(*
Nazwa:			FB_RollerScrewer
Opis:			Zakręcarka rolkowa
Wersja:			v0.5
Data:			2020-03-16
Autor:			DP
Urzadzenia:		Serwo zakręcania, podnosnik JIESANG, rolki, docisk z góry
Konfiguracja:	
Info:  
- ZMIANA ESTOP - blad w trybie manualnym po ESTOPIE
- Dddano kasowanie ruchów w górę po błędzie
- Dodano opisy błędów serwa
- Dodano błędy od nastaw powyżej max i min (error 7 i 8)
- Zmiana Homingów według CatchStation
- zmiana momentu zacisniecia rolek
*)

FUNCTION_BLOCK FB_RollerScrewer
VAR_INPUT
	bEnable:BOOL;						//Zezowlenie na pracę zakręcarki rolkowej
	bEStop:BOOL;						//Stop awaryjny nieaktywny
	bRun:BOOL;							//Rozkaz zakręcania 
	bHoming:BOOL;						//Zezwolenie na wykonanie bazowania i pozycjonowania zakręcarki rolkowej
	bHeightSet:BOOL;					//Ustaw wysokość
	bIgnoreError:BOOL;					//Ignorowania błędów cyklu pracy
	bReset:BOOL;						//Reset błędu, jeśli w stanie "eError"
	nPositionHeightSV:LREAL;			//Wysokość zadana na której ma znajdować się zakręcarka rolkowa
	lrMaxHeight:LREAL;					//Maksymalna wysokość zakręcarki rolkowej
	lrMinHeight:LREAL;					//Minimalna wysokość zakręcarki rolkowej
	iScrewerSetTorque:INT;				//Zadany moment dokręcania [%]
	iScrewTightTime:INT;				//Czas przytrzymania po uzyskaniu momentu [ms] 
	lrScrewerAcceleration:LREAL;			//Przyspieszenie zakręcarki rolkowej
	lrScrewerDeceleration:LREAL;			//Opóźnienie zakręcarki rolkowej
	lrScrewerSpeed:LREAL;				//Prędkość zakręcarki rolkowej
	lrFindigScrewDegree:LREAL;			//Kąt wycofania zakręcarki rolkowej przy szukaniu gwintu
	lrScrewerFrontActualTorque:LREAL;			//Aktualny moment [%]
	lrScrewerRearActualTorque:LREAL;			//Aktualny moment [%]
	rRearActualMotorTemperature :REAL;	// Aktualna temperatura silnika tylniego
	rFrontActualMotorTemperature :REAL;	// Aktualna temperatura silnika tylniego
	bRollsPressedSensor: BOOL; 			// Wejście czujnika zaciśnięcie rolek zakręcarki
	bRollsUnPressedSensor: BOOL; 		// Wejście czujnika odpuszczenia rolek zakręcarki
	bUnPressedTopSensor: BOOL;			// Wejscie czujnika wycofania docisku górnego zakręcarki rolkowej
	lrManualOverride:LREAL;				// Procentowa redukcja prędkości wszystkich serw (Tylko w trybie manualnym)
	bManualMovement:BOOL; 			// Uruchomienie trybu ruchów ręcznych
	bFindingScrewBeginingOption:BOOL; 	//OPCJA. Szukaj początku gwintu nakrętki i opakowania. Zakręcarka napjpierw obraca się w lewo, a po znalezienu gwintu przystepuje do zakręcania;
	nTopActuatorTimeDelayOff:UINT;  	//czas po którym odpusczany jest docisk górny
	bUnlockColision:BOOL:=FALSE;		//Odblokowywanie możliwośći kolizji

	_HEIGHTMOTOR_ :BOOL;	
	bHeightMotorEncoderPulse :BOOL;			//Sygnał impulsów enkodera siłownika
	rHeightMotorPositionOffset :REAL;		//Wysokość bazowani podnośnika
	
	_ALARMINFO_ :BOOL;
	iStationIndex:UDINT;				//Numer stacji 
	sStationName:STRING;				//Nazwa stacji	
	
END_VAR
VAR_OUTPUT
	eState: E_Station;				// Stan zakręcarki rolkowej
	eRunningState:E_RollerScrewer;	// Stan zakręcarki	
	bError: BOOL;					// Błąd stacji
	udiErrorID: UDINT;				// Nr błędu zakręcarki rolkowej
	sErrorDescription:STRING(200);	// Opis błędu
	sErrorDescription2: STRING(200);// Opis błędu
	sErrorStationName: STRING;		// Nazwa stacj
	nScrewingServoErrorNr: UDINT;	// Nr błędu serwo zakręcarki
	bPressingTopActuator: BOOL; 	// Sterowanie zaworem dociskania nakrętki zaciskarki rolkowej od góry
	bPressingRollsActuator: BOOL; 	// Sterowanie zaworem dociskania rolek od boku
	bHeightMotorUp:BOOL;			// Sterowanie silnikiem podnośnika  - RUCH W GÓRĘ
	bHeightMotorDown:BOOL;			// Sterowanie silnikiem podnośnika  - RUCH W DÓŁ
	lrHeightMotorCV:LREAL;			// Aktualna pozycja podnośnika
	uiScrewingFrontTorqueControl:UINT;	// Kontola momentu zakręcania	
	uiScrewingRearTorqueControl:UINT;	// Kontola momentu zakręcania	

	bWarning: BOOL;
	udiWarningID: UDINT;
	tCycleTime:TIME;		
	bHomingDone:BOOL;				// Wymagane ponowne bazowanie (blad podczas bazowania lub stop awaryjny)
	bCycleDone:BOOL;
	bCycleNotDone:BOOL;		
	bAdjustingTorqueDone:BOOL;
	iAdjustingTorque:INT;
	lrAdjustingMaxTorque: LREAL;
END_VAR

VAR
	tonHeightNoChange: TON; // Timer wykrycia braku ruchu siłownika zmiany wysokości stacji
	nLastPositionHeightCV: LREAL;// Pozycja podnośnika w poprzednim cyklu programu
	tonErrorHeightChange: TON; // Timer błędu podnośnika
	rtEncoderHomed:R_TRIG;
	tonCycleTimer:TON;
	rtrigCycleTimerRead:R_TRIG;
	
	mcScrewerFrontMoveVelocity		:MC_MoveVelocity; 	// Ruch prędkościowy
	mcScrewerFrontHalt				:MC_HALT; 			// Zatrzymanie zakręcania
	mcScrewerFrontManualMove		:MC_JOG; 			// Blok obrotu ręcznego zakręcarką
	mcScrewerFrontStop				:MC_Stop; 			// Trwałe zatrzymywanie Serwo
	mcScrewerFrontPower				:MC_POWER; 			// Zasilanie napędu zakręcarki
	fbScrewerFrontHardReset			:FB_SoEReset;
	mcScrewerFrontSoftReset			:MC_Reset;
	mcScrewerFrontSetPosition		:MC_SetPosition;
	mcScrewerFrontMoveRelative		:MC_MoveRelative;

	mcScrewerRearMoveVelocity		:MC_MoveVelocity; 	// Ruch prędkościowy
	mcScrewerRearHalt				:MC_HALT; 			// Zatrzymanie zakręcania
	mcScrewerRearManualMove			:MC_JOG; 			// Blok obrotu ręcznego zakręcarką
	mcScrewerRearStop				:MC_Stop; 			// Trwałe zatrzymywanie Serwo
	mcScrewerRearPower				:MC_POWER; 			// Zasilanie napędu zakręcarki
	fbScrewerRearHardReset			:FB_SoEReset;
	mcScrewerRearSoftReset			:MC_Reset;
	mcScrewerRearSetPosition		:MC_SetPosition;
	mcScrewerRearMoveRelative		:MC_MoveRelative;
	
	bScrewFound: BOOL; //Zakręcarka znalazła początek gwintu
	nMaxTorque: LREAL; //Maksymalny moment podczas szukania poczatku gwintu
	nMinTorque: LREAL; // Najmniejszy moment podczas szukania poczatku gwintu

	tonTightScrewingTimer: TON; // Timer potwierdzenia dokręcenia nakrętki
	bScrewed: BOOL; // Nakrętka zakręcona

	tonTooLongScrewing: TON; // Błąd zbyt długiego zakręcania

	bScrewerFrontServoPower: BOOL; // Zmienna sterujaca zasilaniem serwo Zakręcark
	bScrewerRearServoPower: BOOL; // Zmienna sterujaca zasilaniem serwo Zakręcark

	// Za długie szukanie gwintu
	tonTooLongFinding: TON;
	tonPosDiffError	:TON;
	bStopped: BOOL;
	// Ustawianie pozycji napedu zakrecającego po zakręceniu nakrętki


	// Pozycja rozpoczęcia zakrecania
	lrStartScrewingPos: LREAL;
	
	// Ruch relatywny zakręcarki

	lrStartPositionScrewerFront: LREAL;
	lrStartPositionScrewerRear: LREAL;	
	tonPressingTopDelay: TON;
	tonPressingRollsDelay: TON;
	tonUpPressRollsDelay: TON;
	tonPressingRollsReliseDelay: TON;
	tonTopActuatorDelayOff: TON;
	tonPushingCapDelay: TON;
	tonRollsPressedDelay: TON;
	tofMotorUpPermition: TOF;
	tofMotorDownPermition: TOF;
	tonLimitPosMinReachedDelay: TON;
	tonLimitPosMaxReachedDelay: TON;
	tonMaxHeight: TON;

	bStateError: BOOL;

	//Podnośnik Jiesang	
	fbHeightMotorEncoder			:FB_JiesangActuatorEncoder;	// Blok enkodera podnośnika chwytaka stabilizującego pod zakręcarką	
	bHeightMotorEncoderCounterReset	:BOOL; 						// Sygnał resetu enkodera
	bHeightMotorEncoderHomed		:BOOL;						// Informacja od enkodera że jest zbazowany

	eLastState						:E_Station;			// Stan ogólny bloku
	eLastRunningState				:E_RollerScrewer;	// Stan podbloku
	eLastStateTemp					:E_Station;			// Stan ogólny bloku
	eLastRunningStateTemp			:E_RollerScrewer;	// Stan podbloku	
	sWarningDescription				:STRING;
	
	nCaseAdjustingTorque: INT;
	tonAdjustingTightScrewingTimer: TON;
	tonAdjustingGripperClose: TON;
	uiAdjustingScrewerTorqueControl: UINT;
	bAdjustingScrewed: BOOL;
	tonAdjustingCase40: TON;
	bAdjustingSetTorqueAchieved: BOOL;
	bAdjustingTorqueTooHigh: BOOL;
	bAdjustingTorqueTooLow: BOOL;
	lrMotorNominalTorque: LREAL;
	lrScrewerActualTorqueNm: LREAL;
	
	tonDelayServoOn			: TON;

	tonRearActualMotorTemperatureTooHigh: TON;
	tonFrontActualMotorTemperatureTooHigh: TON;
END_VAR

VAR_IN_OUT
	bManualPressingTopActuator		:BOOL;		// Sterowanie w trybie serwisowym zaworem dociskania nakrętki zaciskarki rolkowej od góry
	bManualPressingRollsActuator	:BOOL;		// Sterowanie w trybie serwisowym zaworem dociskania rolek od boku
	bManualHeightMotorUp			:BOOL;		// Ruch ręczny podnośnika stacji w górę
	bManualHeightMotorDown			:BOOL;		// Ruch ręczny podnośnika stacji w dół
	bManualScrewClockwise			:BOOL;		// Ruch ręczny zakręcarką w kierunku wskazówek zegara;
	bManualScrewCClockwise			:BOOL;		// Ruch ręczny zakręcarką w kierunku przeciwnym do wskazówek zegara;
	RollerScrewerFrontAxisRef		:AXIS_REF;	// Struktura sterowania NC dla serwa zakręcania
	RollerScrewerRearAxisRef		:AXIS_REF;	// Struktura sterowania NC dla serwa zakręcania	

END_VAR

(*Przepisywanie Homingu , rozdzielenie wyjść*)

HeightMotor();
ErrorHandling();
Control();
ServoFrontControlBlocks();
ServoRearControlBlocks();
Statistics();

(*Zapisywanie ostatniego stanu*)
IF eLastStateTemp<>eState THEN
	eLastState := eLastStateTemp;
END_IF
eLastStateTemp := eState;
IF eLastRunningStateTemp<>eRunningState THEN
	eLastRunningState := eLastRunningStateTemp;
END_IF
eLastRunningStateTemp := eRunningState;
(*Koniec Zapisywanie ostatniego stanu*)


nLastPositionHeightCV:=lrHeightMotorCV;

ACTION Control:
	(** TIMERY**)
	rtEncoderHomed				(CLK:= bHeightMotorEncoderHomed,Q=>);
	tonHeightNoChange			(IN:= ((bHeightMotorUp OR bHeightMotorDown) AND (nLastPositionHeightCV=lrHeightMotorCV)), PT:= T#1S); 
	tonLimitPosMinReachedDelay	(IN:= (lrHeightMotorCV<=lrMinHeight) AND eState=E_Station.eHoming,PT:= T#2S);
	tonLimitPosMaxReachedDelay	(IN:= (lrHeightMotorCV>=lrMaxHeight) AND eState=E_Station.eHoming,PT:= T#2S);

	tonPressingRollsReliseDelay(IN:= NOT bPressingRollsActuator AND NOT bPressingTopActuator, PT:= T#40MS);	
	tonTightScrewingTimer		(IN:= (eRunningState=E_RollerScrewer.eScrewing) AND 
								NOT tonTightScrewingTimer.Q AND mcScrewerFrontMoveVelocity.Execute AND mcScrewerRearMoveVelocity.Execute AND 
								((lrScrewerFrontActualTorque>=iScrewerSetTorque) OR (lrScrewerRearActualTorque>=iScrewerSetTorque)) AND 
								ABS(RollerScrewerFrontAxisRef.NcToPlc.PosDiff)>360 AND ABS(RollerScrewerRearAxisRef.NcToPlc.PosDiff)>360 
								AND NOT bScrewed ,PT:= INT_TO_TIME(iScrewTightTime));
	tonTopActuatorDelayOff		(IN:= bPressingTopActuator AND eRunningState=E_RollerScrewer.eScrewing, PT:= UINT_TO_TIME(nTopActuatorTimeDelayOff));	
	tonPushingCapDelay			(IN:= (eRunningState=E_RollerScrewer.ePushingCap) AND (NOT bUnPressedTopSensor OR  nTopActuatorTimeDelayOff=0), PT:= T#100MS);
	tonRollsPressedDelay		(IN:= (eRunningState=E_RollerScrewer.ePushingCap) AND NOT bRollsUnpressedSensor, PT:= T#0MS); //bylo 200

	tonDelayServoOn				(IN:=(eState = E_Station.ePreparingToReady), PT:=T#2S);
	
	(*****Wyłączenie enable*****)
	IF NOT bEnable THEN
		IF eState <> E_Station.eDisabled AND eState <> E_Station.ePreparingToDisable THEN
				eState 								:= E_Station.ePreparingToDisable; 
		END_IF	
	END_IF

	(*****Estop*****)
	IF NOT bEstop  THEN	
		IF eState <> E_Station.eAborted AND eState <> E_Station.eAborting AND eState <> E_Station.eDisabled THEN
				eState 								:= E_Station.eAborting; 
		END_IF
	END_IF

	
	CASE eState OF
	/////////////////////////////	
		E_Station.eDisabled: 						// Stan nieaktywnosci (Stacja wyłączona) 
		
			IF bEnable THEN
				eState 								:= E_Station.ePreparingToReady; 
			END_IF 
			
    /////////////////////////////	    
		E_Station.eAborted: 						// Stan bezpiecznego zatrzymania (po Abortingu) 

			IF bEStop THEN
				eState 								:= E_Station.ePreparingToReady;
			END_IF
			
	/////////////////////////////	
		E_Station.eAborting:                 		// Stan bezpiecznego zatrzymywania (po EStopie)
		
			bHeightMotorDown		:=	FALSE;
			bHeightMotorUp			:=	FALSE;	
		
			bPressingTopActuator					:= FALSE;
			bPressingRollsActuator					:= FALSE;

			mcScrewerFrontPower.Override			:= 100;
			mcScrewerFrontStop.Execute				:= NOT bStopped;
			mcScrewerFrontMoveVelocity.Execute		:= FALSE;
			mcScrewerFrontManualMove.JogBackwards	:= FALSE;
			mcScrewerFrontManualMove.JogForward		:= FALSE;
			
			mcScrewerRearPower.Override				:= 100;
			mcScrewerRearStop.Execute				:= NOT bStopped;
			mcScrewerRearMoveVelocity.Execute		:= FALSE;
			mcScrewerRearManualMove.JogBackwards	:= FALSE;
			mcScrewerRearManualMove.JogForward		:= FALSE;
			
			IF ((mcScrewerFrontStop.Done OR NOT bScrewerFrontServoPower) AND (mcScrewerRearStop.Done OR NOT bScrewerRearServoPower)) OR bStopped THEN
				bStopped							:= FALSE;
				bScrewerFrontServoPower				:= FALSE;
				mcScrewerFrontStop.Execute			:= FALSE;
				bScrewerRearServoPower				:= FALSE;
				mcScrewerRearStop.Execute			:= FALSE;
				eState								:= E_Station.eAborted; 
				eRunningState						:= E_RollerScrewer.eReady;
			END_IF		
			
			
	/////////////////////////////			
		E_Station.eError:                 	 		// Stan błędu 	
				
			IF bReset THEN
				eState 								:= E_Station.eResetting;
			ELSE
				mcScrewerFrontSoftReset				(Execute:= FALSE,Axis:= RollerScrewerFrontAxisRef);	
				mcScrewerRearSoftReset				(Execute:= FALSE,Axis:= RollerScrewerRearAxisRef);	
			END_IF
			
	/////////////////////////////
		E_Station.eResetting:						// Stan resetowania bledu (po Errorze)
			
			//Procedura obsługi resetu w zależności od błędu
			CASE udiErrorID-iStationIndex OF
		
				//Error 1 - ZA DŁUGIE ZAKRĘCANIE	
				1:
					IF tonPressingRollsReliseDelay.Q AND RollerScrewerFrontAxisRef.Status.StandStill AND RollerScrewerRearAxisRef.Status.StandStill THEN
						;
						udiErrorID					:= 0;
						sErrorDescription			:= '';	
						bError 						:= FALSE;	
					END_IF
					
				//Error 2,4,5,6,7,8	
				2,4,5,6,7,8:   
					 bError 						:= FALSE;
					 udiErrorID						:= 0;
					 sErrorDescription				:= '';		
			
				//Error 3 - BŁĄD SERWA ZAKRĘCANIA
				3:	
					//fbScrewerHardReset			(Execute:= NOT mcHeightMoveAbsolute.Execute,Axis:= ScrewingAxisRef);
					mcScrewerFrontSoftReset			(Execute:= TRUE,Axis:= RollerScrewerFrontAxisRef);
					mcScrewerRearSoftReset			(Execute:= TRUE,Axis:= RollerScrewerRearAxisRef);
					IF NOT fbScrewerFrontHardReset.Busy AND NOT mcScrewerFrontSoftReset.Busy AND mcScrewerFrontPower.Status AND NOT RollerScrewerFrontAxisRef.Status.Error
					AND NOT fbScrewerRearHardReset.Busy AND NOT mcScrewerRearSoftReset.Busy AND mcScrewerRearPower.Status AND NOT RollerScrewerRearAxisRef.Status.Error  THEN
						fbScrewerFrontHardReset		(Execute:= FALSE,Axis:= RollerScrewerFrontAxisRef);
						fbScrewerRearHardReset		(Execute:= FALSE,Axis:= RollerScrewerRearAxisRef);
						mcScrewerFrontSoftReset		(Execute:= FALSE,Axis:= RollerScrewerFrontAxisRef);
						mcScrewerRearSoftReset		(Execute:= FALSE,Axis:= RollerScrewerRearAxisRef);
						bError 						:= FALSE;
						udiErrorID					:= 0;
						nScrewingServoErrorNr		:= 0;
						mcScrewerFrontPower.Override:= 100;
						mcScrewerRearPower.Override	:= 100;
						eState						:= E_Station.eReady;
						sErrorDescription			:= '';	
			
					ELSIF NOT fbScrewerFrontHardReset.Busy AND NOT mcScrewerFrontSoftReset.Busy AND NOT mcScrewerFrontPower.Status AND NOT bScrewerFrontServoPower AND NOT RollerScrewerFrontAxisRef.Status.Error
						AND NOT fbScrewerRearHardReset.Busy AND NOT mcScrewerRearSoftReset.Busy AND NOT mcScrewerRearPower.Status AND NOT bScrewerRearServoPower AND NOT RollerScrewerRearAxisRef.Status.Error THEN
						//fbScrewerHardReset(Execute:= FALSE,Axis:= ScrewingAxisRef);
						mcScrewerFrontSoftReset		(Execute:= FALSE,Axis:= RollerScrewerFrontAxisRef);
						mcScrewerRearSoftReset		(Execute:= FALSE,Axis:= RollerScrewerRearAxisRef);
						udiErrorID					:= 0;
						nScrewingServoErrorNr		:= 0;
						mcScrewerFrontPower.Override:= 100;
						mcScrewerRearPower.Override	:= 100;
						bError 						:= FALSE;
						sErrorDescription			:= '';
					END_IF		
					
			END_CASE	
			
			IF NOT bError THEN
				udiErrorID 							:= 	0;
   				sErrorDescription 					:= 	'';
	                                				
				eState 								:= 	E_Station.ePreparingToReady;
				mcScrewerFrontStop.Execute			:= FALSE;    
				mcScrewerRearStop.Execute			:= FALSE; 
			ELSE                    	
				eState 								:= 	E_Station.eError;
			END_IF
        
	/////////////////////////////
		E_Station.eManualMovement:     				// Stan ruchów manualnych  
       
			ManualMovements();
			//Wyjście z trybu serwisowego
			IF NOT bManualMovement THEN
				bManualPressingTopActuator			:= 	FALSE;
				bManualPressingRollsActuator		:= 	FALSE;
				bHeightMotorUp						:= 	FALSE;
				bHeightMotorDown					:= 	FALSE;
				mcScrewerFrontPower.Override			:= 	100;
				mcScrewerRearPower.Override			:= 	100;
				eState								:= 	E_Station.eReady;
			END_IF

	/////////////////////////////
		E_Station.eHoming:							// Stan bazowania 

			Homing();
			IF NOT bHoming AND NOT bHeightSet THEN
			   eState								:= 	E_Station.ePreparingToReady;
			   bHeightMotorUp						:= 	FALSE;
				bHeightMotorDown					:= 	FALSE;
			END_IF		
			
	/////////////////////////////
		E_Station.eHomingDone:                  	// Stan wykonania bazowania 

			bHeightMotorDown						:= 	FALSE;
			bHeightMotorUp							:= 	FALSE;
			bHeightMotorEncoderCounterReset			:= 	FALSE;
			bHomingDone								:= 	TRUE;
			IF NOT bHoming AND NOT bHeightSet THEN
			   	eState								:= 	E_Station.eReady;
			END_IF
			
	/////////////////////////////
		E_Station.ePreparingToReady:            	// Stan przygotowywania do gotowosci (zawsze przed Ready)  
	
			IF tonDelayServoOn.Q THEN
				bScrewerFrontServoPower				:= 	TRUE;
				bScrewerRearServoPower				:= 	TRUE;
			END_IF	

				
			bPressingTopActuator					:= 	FALSE;
			bPressingRollsActuator					:= 	FALSE;
			IF mcScrewerFrontPower.Status AND mcScrewerRearPower.Status THEN  	
				eState								:= 	E_Station.eReady;
				eRunningState						:= 	E_RollerScrewer.eReady;
			END_IF                              	
         	IF bIgnoreError THEN                	
				eState								:= 	E_Station.eReady;
				eRunningState						:= 	E_RollerScrewer.eReady;
			END_IF
	
	/////////////////////////////
		E_Station.ePreparingToDisable:         	 	// Stan przygotowywania do nieaktywnosci (po wyłączeniu Enable) 
  
			bScrewerFrontServoPower					:= 	TRUE;
			bScrewerRearServoPower					:= 	TRUE;

			
			bPressingTopActuator					:= 	FALSE;
			bPressingRollsActuator					:= 	FALSE;
			                        				
			bHeightMotorUp							:= 	TRUE;
			bHeightMotorDown						:= 	FALSE;
			IF tonHeightNoChange.Q THEN	
				bHeightMotorUp:= FALSE;
				IF  mcScrewerFrontPower.Status THEN
					bScrewerFrontServoPower			:= 	FALSE; //LU205
					bScrewerRearServoPower			:= 	FALSE;;//LU205
					eState							:= 	E_Station.eDisabled;
					eRunningState					:= 	E_RollerScrewer.eReady;
				END_IF
			END_IF				
         	IF bIgnoreError THEN
				bHeightMotorUp						:= 	FALSE;
				eState								:= 	E_Station.eDisabled;
				eRunningState						:= 	E_RollerScrewer.eReady;
			END_IF
			
	/////////////////////////////
		E_Station.eReady:							// Stan gotowosci 
		
			mcScrewerFrontStop.Execute:= FALSE;
		
			IF bRun AND NOT bCycleDone AND NOT bCycleNotDone THEN
				eState 								:= E_Station.eStarting; 
			END_IF
			IF bHoming OR bHeightSet THEN
				eState 								:= E_Station.eHoming; 
			END_IF
			IF bManualMovement THEN
				//Jeśli przejście w tryb ruchów manualnych przepisz wszystkie stany siłowników sterowanych przez moduł
				//aby zapobiec ewentualnym kolizjom po wejściu w tryb serwisowy
				bManualPressingTopActuator			:= 	bPressingTopActuator;
				bManualPressingRollsActuator		:= 	bPressingRollsActuator;
				bManualHeightMotorUp				:= 	bHeightMotorUp;
				bManualHeightMotorDown				:= 	bHeightMotorDown;
				mcScrewerFrontStop.Execute			:= 	FALSE;
				mcScrewerRearStop.Execute			:= 	FALSE;
				eState 								:= 	E_Station.eManualMovement; 
			END_IF
			IF NOT bRun THEN
				bCycleDone 							:= FALSE;
				bCycleNotDone 						:= FALSE;	
				bWarning							:= FALSE;	
			END_IF      

			bStopped								:= FALSE;
			mcScrewerFrontStop.Execute				:= FALSE;    
			mcScrewerRearStop.Execute				:= FALSE;                   			
			
	/////////////////////////////
		E_Station.eStopping:					// Stan zatrzymywania 
			
			Running();

			bPressingTopActuator					:= 	FALSE;
			bPressingRollsActuator					:= 	FALSE;
			
			mcScrewerFrontHalt.Execute				:= 	FALSE;			
			mcScrewerFrontStop.Execute				:= 	NOT bStopped;
			mcScrewerFrontMoveRelative.Execute		:= 	FALSE;
			mcScrewerFrontMoveVelocity.Execute		:= 	FALSE;
			uiScrewingFrontTorqueControl			:= 	0; // bylo 6000	
			mcScrewerFrontSoftReset					(Axis:= RollerScrewerFrontAxisRef, Execute:= TRUE);

			mcScrewerRearHalt.Execute				:= 	FALSE;			
			mcScrewerRearStop.Execute				:= 	NOT bStopped;
			mcScrewerRearMoveRelative.Execute		:= 	FALSE;
			mcScrewerRearMoveVelocity.Execute		:= 	FALSE;
			uiScrewingRearTorqueControl				:= 	0; // bylo 6000	
			mcScrewerRearSoftReset					(Axis:= RollerScrewerRearAxisRef, Execute:= TRUE);
			
			IF  (mcScrewerFrontStop.Done OR mcScrewerFrontStop.CommandAborted) AND 
				(mcScrewerRearStop.Done OR mcScrewerRearStop.CommandAborted) 
				THEN
				mcScrewerFrontStop.Execute			:= 	FALSE;
				mcScrewerRearStop.Execute			:= 	FALSE;
				bStopped							:= 	FALSE;
				eState 								:= 	E_Station.eReady;
			END_IF
		
		
	/////////////////////////////
		E_Station.eStarting:                  	// Stan uruchamiania (po Ready)
		
			eState									 := E_Station.eRunning; 
			
	/////////////////////////////
		E_Station.eRunning:               		// Stan wykonywania cyklu (po Startingu), w tym stanie osobny
 
			Running();
			IF NOT bRun THEN					(*Przerywanie cyklu*)
				eState 				 				:= E_Station.eStopping;	
			END_IF
			IF bCycleDone OR bCycleNotDone THEN (*Cykl zakończony*)
				eState 								 := E_Station.eReady;
			END_IF	
			
			
	/////////////////////////////		
	END_CASE
END_ACTION

ACTION ErrorHandling:
//OBSŁUGA BŁĘDÓW ZAKRĘCARKI ROLKOWEJ

RollerScrewerFrontAxisRef.ReadStatus();


//**********************LISTA BŁĘDÓW******************************
bStateError:= (eState=E_Station.eError) OR (eState=E_Station.eResetting) OR bIgnoreError;

IF bEnable THEN
	
	//Error 1 - ZA DŁUGIE ZAKRĘCANIE
	tonTooLongScrewing(IN:=(eRunningState=E_RollerScrewer.eScrewing),PT:=T#2S);
	tonTooLongFinding(IN:=(eRunningState=E_RollerScrewer.eFindingScrew),PT:=T#1S500MS);
	tonPosDiffError(IN:=((ABS(RollerScrewerFrontAxisRef.NcToPlc.ActPos-lrStartPositionScrewerFront)>=3080) OR ABS(RollerScrewerRearAxisRef.NcToPlc.ActPos-lrStartPositionScrewerRear)>=3080)  AND eRunningState=E_RollerScrewer.eScrewing,PT:=T#1MS);
	IF (tonTooLongScrewing.Q OR tonTooLongFinding.Q OR tonPosDiffError.Q) AND NOT bStateError THEN
		bHeightMotorUp:=FALSE;
		bHeightMotorDown:=FALSE;
		bStopped:=FALSE;
		bPressingTopActuator:=FALSE;
		bPressingRollsActuator:=FALSE;
		mcScrewerFrontMoveVelocity.Execute:=FALSE;
		mcScrewerFrontHalt.Execute:=FALSE;
		mcScrewerRearMoveVelocity.Execute:=FALSE;
		mcScrewerRearHalt.Execute:=FALSE;
		eState	:= E_Station.eStopping; 
		eRunningState	:=	E_RollerScrewer.eNotDone;
		bWarning:=TRUE;
		udiWarningID := 1;
		udiErrorID := 1;
		udiErrorID := udiErrorID+iStationIndex;
		sWarningDescription:='Przekroczenie czasu zakręcania - zmień ustawienia zakręcania';	
		(*Kasownie momentu po zakręceniu*)		
		uiScrewingFrontTorqueControl:=0; // bylo 6000
		uiScrewingRearTorqueControl:=0; // bylo 6000
		mcScrewerFrontSoftReset(Axis:=RollerScrewerFrontAxisRef, Execute:= TRUE);
		mcScrewerRearSoftReset(Axis:=RollerScrewerRearAxisRef, Execute:= TRUE);
	END_IF
	
	//Error 2 - podnośnik nie porusza się pomimo wysterowania 
	tonErrorHeightChange(IN:=(bHeightMotorUp OR bHeightMotorDown) AND nLastPositionHeightCV=lrHeightMotorCV, PT:=T#3S);
	IF tonErrorHeightChange.Q AND NOT bStateError THEN
		bHeightMotorUp:=FALSE;
		bHeightMotorDown:=FALSE;
		bError := TRUE;
		udiErrorID:=2;
		udiErrorID := udiErrorID+iStationIndex;	
		sErrorDescription:='Blokada podnośnika lub brak zasilania - sprawdź czujnik lub odblokuj mechanicznie';	
	END_IF
	
	//Error 3 - BŁĄD SERWA ZAKRĘCAJĄCEGO
	IF RollerScrewerFrontAxisRef.Status.Error OR mcScrewerFrontStop.Error OR RollerScrewerRearAxisRef.Status.Error OR mcScrewerRearStop.Error AND NOT bStateError THEN
		bHeightMotorUp:=FALSE;
		bHeightMotorDown:=FALSE;
		bStopped:=FALSE;
		bError := TRUE;
		udiErrorID:=3;
		udiErrorID := udiErrorID+iStationIndex;	
		nScrewingServoErrorNr:=RollerScrewerFrontAxisRef.Status.ErrorID;
		sErrorDescription:='Błąd napędu zakręcającego. Błąd NC:';
		sErrorDescription2:=F_AxErrMsg(nScrewingServoErrorNr);
	END_IF;
	
	//Error 4 - BLAD DOCISKU NAKRĘTKI OD GÓRY ZAKRECARKI
	tonPressingTopDelay(IN:=(NOT bPressingTopActuator AND NOT bUnPressedTopSensor),PT:=T#1S);
	IF tonPressingTopDelay.Q AND NOT bStateError THEN
		bHeightMotorUp:=FALSE;
		bHeightMotorDown:=FALSE;
		bPressingTopActuator:=FALSE;
		bError := TRUE;
		udiErrorID:=4;
		udiErrorID := udiErrorID+iStationIndex;			
		sErrorDescription:='Błąd docisku nakrętki od góry - sprawdź czujnik ';
	END_IF;
	
	//Error 5 - BLAD DOCISKU ROLEK DOCISKAJĄCYCH ZAKRECARKI
	tonPressingRollsDelay(IN:=(bPressingRollsActuator AND NOT bRollsPressedSensor),PT:=T#1S);
	IF tonPressingRollsDelay.Q AND NOT bStateError THEN
		bHeightMotorUp:=FALSE;
		bHeightMotorDown:=FALSE;
		bPressingRollsActuator:=FALSE;
		bError := TRUE;
		udiErrorID:=5;
		udiErrorID := udiErrorID+iStationIndex;			
		sErrorDescription:='Błąd docisku rolek - sprawdź czujnik';
	END_IF;
	
	//Error 6 - BLAD ODPUSZCZENIA ROLEK DOCISKAJĄCYCH ZAKRECARKI
	tonUpPressRollsDelay(IN:=(NOT bPressingRollsActuator AND NOT bRollsUnPressedSensor),PT:=T#1S);
	IF tonUpPressRollsDelay.Q AND NOT bStateError  THEN
		bHeightMotorUp:=FALSE;
		bHeightMotorDown:=FALSE;
		bPressingRollsActuator:=FALSE;
		bError := TRUE;
		udiErrorID:=6;
		udiErrorID := udiErrorID+iStationIndex;			
		sErrorDescription:='Błąd odocisku rolek - sprawdź czujnik';
	END_IF;
	
	//Error 7 - Bład nastaw max
	tonMaxHeight(IN:=nPositionHeightSV>lrMaxHeight AND NOT bHomingDone AND eState=E_Station.eReady,PT:=T#30S);
	IF tonMaxHeight.Q AND NOT bStateError  THEN
		bHeightMotorUp:=FALSE;
		bHeightMotorDown:=FALSE;
		bError := TRUE;
		udiErrorID:=7;
		udiErrorID := udiErrorID+iStationIndex;			
		sErrorDescription:='Wartość zadana wysokości jest większa od maksymalnej - zmień ustawienia w recepturze';
		sErrorDescription2:=REAL_TO_STRING(LREAL_TO_INT(lrMaxHeight));
	END_IF
	
	//Error 8 - ZBYT WYSOKA TEMPERATURA SILNIKA TYLNIEGO
	tonRearActualMotorTemperatureTooHigh(IN:=rRearActualMotorTemperature>130, PT:=T#10S);
	IF tonRearActualMotorTemperatureTooHigh.Q AND NOT bStateError THEN
		bHeightMotorUp:=FALSE;
		bHeightMotorDown:=FALSE;
		bStopped:=FALSE;
		bError := TRUE;
		udiErrorID	:=	8;
		udiErrorID	:=	udiErrorID+iStationIndex;
		sErrorDescription:='Zbyt wysoka temperatura napędu zakręcającego tylniego > 130C - zmniejsz moment zakręcania';
		sErrorDescription2:=INT_TO_STRING(REAL_TO_INT(rRearActualMotorTemperature));
	END_IF
	
	//Error 9 - ZBYT WYSOKA TEMPERATURA SILNIKA PRZEDNIEGO
	tonFrontActualMotorTemperatureTooHigh(IN:=rFrontActualMotorTemperature>130, PT:=T#10S);
	IF tonFrontActualMotorTemperatureTooHigh.Q AND NOT bStateError THEN
		bHeightMotorUp:=FALSE;
		bHeightMotorDown:=FALSE;
		bStopped:=FALSE;
		bError := TRUE;
		udiErrorID	:=	9;
		udiErrorID	:=	udiErrorID+iStationIndex;
		sErrorDescription:='Zbyt wysoka temperatura napędu zakręcającego przedniego > 130C - zmniejsz moment zakręcania';
		sErrorDescription2:=INT_TO_STRING(REAL_TO_INT(rFrontActualMotorTemperature));
	END_IF 	
ELSE
	bError := FALSE;	
END_IF

//******************PRZEJŚCIE DO eERROR*****************************

IF bError AND NOT bStateError THEN
	IF eLastState = eRunning THEN
		bCycleNotDone := TRUE;
	END_IF
	eState := E_Station.eError;
END_IF

//****************WYŚWIETLANIE STATUSU BLEDU***********************

(*Wyświetlanie błedu na wyjściu*)
bError;

(*Przepisywanie nazwy stacji*)
sErrorStationName := sStationName;
END_ACTION

ACTION HeightMotor:
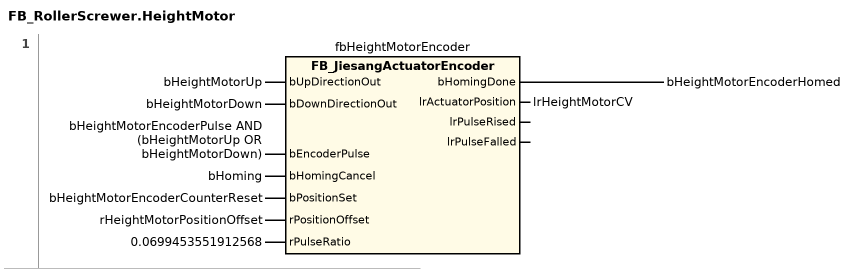
// NETWORK 1
fbHeightMotorEncoder(
    bUpDirectionOut := bHeightMotorUp,
    bDownDirectionOut := bHeightMotorDown,
    bEncoderPulse := bHeightMotorEncoderPulse AND (bHeightMotorUp OR bHeightMotorDown),
    bHomingCancel := bHoming,
    bPositionSet := bHeightMotorEncoderCounterReset,
    rPositionOffset := rHeightMotorPositionOffset,
    rPulseRatio := 0.0699453551912568,
    lrActuatorPosition => lrHeightMotorCV); // FB_JiesangActuatorEncoder
bHeightMotorEncoderHomed := fbHeightMotorEncoder.bHomingDone;
END_ACTION

ACTION Homing:
//BAZOWANIE
bPressingTopActuator:=FALSE;
bPressingRollsActuator:=FALSE;
	
//Podnoszenie stacji do maksymalnej pozycji
IF NOT bHeightMotorEncoderHomed OR rtEncoderHomed.Q THEN
	
	//Wylaczanie serwa zakręcania podczas bazowania
	mcScrewerFrontPower.Override:=100;
	mcScrewerFrontStop.Execute:=NOT bStopped;
	mcScrewerFrontMoveVelocity.Execute:=FALSE;
	mcScrewerFrontManualMove.JogBackwards:=FALSE;
	mcScrewerFrontManualMove.JogForward:=FALSE;
	
	mcScrewerRearPower.Override:=100;
	mcScrewerRearStop.Execute:=NOT bStopped;
	mcScrewerRearMoveVelocity.Execute:=FALSE;
	mcScrewerRearManualMove.JogBackwards:=FALSE;
	mcScrewerRearManualMove.JogForward:=FALSE;
	
	bHeightMotorUp:=TRUE;
	bHeightMotorDown:=FALSE;
	IF tonHeightNoChange.Q THEN
		bHeightMotorEncoderCounterReset:=TRUE;
		bHeightMotorUp:=FALSE;
    END_IF
	//Jesli enkoder zbazowany zakończ bazowanie	
	IF rtEncoderHomed.Q THEN
		bHeightMotorUp:=FALSE;
		bHeightMotorDown:=FALSE;
		eState:=E_Station.eHomingDone;
	END_IF		
		
//Po podniesieniu stacji opuszczanie do ustalonej wysokości
ELSIF bHeightMotorEncoderHomed THEN
	bHeightMotorEncoderCounterReset:=FALSE;
	bHeightMotorUp:=lrHeightMotorCV<=nPositionHeightSV;
	bHeightMotorDown:=lrHeightMotorCV>=nPositionHeightSV;
	//Kiedy stacja osiągnie wysokość zadaną
	IF ABS(lrHeightMotorCV-nPositionHeightSV)<1 OR tonLimitPosMaxReachedDelay.Q OR tonLimitPosMinReachedDelay.Q THEN
		bHeightMotorDown:=FALSE;
		bHeightMotorUp:=FALSE;
		eState:=E_Station.eHomingDone;
	END_IF			
END_IF
END_ACTION

ACTION ManualMovements:

//W trybie ruchów manualnych wykonuj ruchy za pomocą rozkazów manualnych
IF NOT bRun THEN
	mcScrewerFrontPower.Override:=lrManualOverride;
	uiScrewingFrontTorqueControl:=(INT_TO_UINT(iScrewerSetTorque+5)*10)*BOOL_TO_UINT(bManualScrewClockwise OR bManualScrewCClockwise);
	mcScrewerFrontManualMove.JogForward:=bManualScrewClockwise;	
	mcScrewerFrontManualMove.JogBackwards:=bManualScrewCClockwise;

	mcScrewerRearPower.Override:=lrManualOverride;
	uiScrewingRearTorqueControl:=(INT_TO_UINT(iScrewerSetTorque+5)*10)*BOOL_TO_UINT(bManualScrewClockwise OR bManualScrewCClockwise);
	mcScrewerRearManualMove.JogForward:=bManualScrewClockwise;	
	mcScrewerRearManualMove.JogBackwards:=bManualScrewCClockwise;
	
	bPressingTopActuator:=bManualPressingTopActuator;
	bPressingRollsActuator:=bManualPressingRollsActuator;
	bHeightMotorUp:=bManualHeightMotorUp;
	bHeightMotorDown:=bManualHeightMotorDown;
ELSE	//Kasuje zeby po cyklu nic sie nie poruszało
	bManualPressingTopActuator:=FALSE;
	bManualPressingRollsActuator:=FALSE;
	bManualHeightMotorUp  := FALSE;
	bManualHeightMotorDown  := FALSE;
END_IF


IF bHoming OR bHeightSet THEN
	eState:=E_Station.eHoming;
END_IF


Running();

	
//Zabezpieczenie przed kolizją stacji poprzez ruch podnośnika	
IF bHeightMotorDown AND lrHeightMotorCV<=lrMinHeight AND NOT bHoming AND NOT bHeightSet THEN
	bHeightMotorDown:=FALSE;
END_IF	

IF bHeightMotorUp AND lrHeightMotorCV>=lrMaxHeight AND NOT bHoming AND NOT bHeightSet THEN
	bHeightMotorUp:=FALSE;
END_IF		 

IF NOT bRun THEN
	bCycleDone 					:= FALSE;
	bCycleNotDone 				:= FALSE;
	bWarning					:= FALSE;		
END_IF
END_ACTION

ACTION Running:
//Timery
tofMotorUpPermition(IN:=bHeightMotorDown, PT:=T#250MS);
tofMotorDownPermition(IN:=bHeightMotorUp, PT:=T#250MS);	

CASE eRunningState OF

//====================================

	//Niegotowy
	E_RollerScrewer.eDisabled:
		eRunningState:=E_RollerScrewer.eReady;
	
	(*Oczekiwanie na wykonanie pojedynczego cyklu*)
	E_RollerScrewer.eReady:
        mcScrewerFrontSoftReset								(Axis:=RollerScrewerFrontAxisRef, Execute:=FALSE);                                       	
		mcScrewerFrontMoveVelocity.Execute					:=	FALSE;
		uiScrewingFrontTorqueControl						:=	6000; 
		
		mcScrewerRearSoftReset								(Axis:=RollerScrewerRearAxisRef, Execute:=FALSE);                                       	
		mcScrewerRearMoveVelocity.Execute					:=	FALSE;
		uiScrewingRearTorqueControl							:=	6000;    
		
		bScrewed											:=	FALSE;
		bScrewFound											:=	FALSE;
		tonTightScrewingTimer(IN:=FALSE,PT:=INT_TO_TIME(iScrewTightTime));                                           	
		IF NOT bCycleDone AND NOT bCycleNotDone THEN                                           	
			IF bRun THEN                	
				eRunningState							:=	E_RollerScrewer.ePushingCap;	
			END_IF
		END_IF


//====================================
	
		
	//ZAKRĘCARKA W STANIE WCISKANIA NAKRĘTKI
	E_RollerScrewer.ePushingCap:
			//ZRozkaz wciskania nakrętki od góry
			bPressingTopActuator:=nTopActuatorTimeDelayOff>0;
			//bPressingTopActuator:=TRUE;
			bPressingRollsActuator:=tonPushingCapDelay.Q; //zmiana1
			//Jeśli znikł czujnik wycofania docisku to przejdz dalej
			IF (NOT bUnPressedTopSensor OR nTopActuatorTimeDelayOff=0) AND bRollsPressedSensor AND tonRollsPressedDelay.Q THEN
				eRunningState:=E_RollerScrewer.ePushed;
			END_IF
			

		
//====================================		
				
	E_RollerScrewer.ePushed:
	
		IF bFindingScrewBeginingOption THEN
			mcScrewerFrontMoveRelative.Execute				:=	TRUE;
			mcScrewerFrontMoveRelative.Velocity				:=	lrScrewerSpeed;
			mcScrewerRearMoveRelative.Execute				:=	TRUE;
			mcScrewerRearMoveRelative.Velocity				:=	lrScrewerSpeed;			
			uiScrewingFrontTorqueControl						:=	4000;
			uiScrewingRearTorqueControl						:=	4000;
		END_IF
		mcScrewerFrontMoveVelocity.Velocity					:=	lrScrewerSpeed;
		mcScrewerRearMoveVelocity.Velocity					:=	lrScrewerSpeed;
		IF bFindingScrewBeginingOption THEN		
			eRunningState								:=	E_RollerScrewer.eFindingScrew;
			nMaxTorque									:=	0;
			nMinTorque									:=	2000;
			bScrewFound									:=	FALSE;	
		ELSE
			lrStartPositionScrewerFront					:=	RollerScrewerFrontAxisRef.NcToPlc.ActPos;
			lrStartPositionScrewerRear					:=	RollerScrewerRearAxisRef.NcToPlc.ActPos;
			eRunningState								:=	E_RollerScrewer.eScrewing;
			mcScrewerFrontMoveVelocity.Execute				:=	TRUE;
			mcScrewerRearMoveVelocity.Execute				:=	TRUE;
			lrStartScrewingPos							:=	RollerScrewerFrontAxisRef.NcToPlc.ActPos;		
		END_IF
			
	
//====================================					
	
	E_RollerScrewer.eFindingScrew:
	
			mcScrewerFrontMoveRelative.Execute				:=	TRUE;
			mcScrewerFrontMoveRelative.Velocity				:=	lrScrewerSpeed;
			mcScrewerRearMoveRelative.Execute				:=	TRUE;
			mcScrewerRearMoveRelative.Velocity				:=	lrScrewerSpeed;
			uiScrewingFrontTorqueControl					:=	4000;
			uiScrewingRearTorqueControl						:=	4000;	
			IF (mcScrewerFrontMoveRelative.Done AND mcScrewerRearMoveRelative.Done) OR bScrewFound THEN
			
				mcScrewerFrontMoveRelative.Execute			:=	FALSE;
				mcScrewerRearMoveRelative.Execute			:=	FALSE;
				bScrewFound									:=	TRUE;
				mcScrewerFrontHalt.Execute					:=	FALSE;
				mcScrewerRearHalt.Execute					:=	FALSE;	
				eRunningState								:=	E_RollerScrewer.eScrewing;
			
				mcScrewerFrontMoveVelocity.Execute			:=	TRUE;
				mcScrewerRearMoveVelocity.Execute			:=	TRUE;
				lrStartPositionScrewerFront					:=	RollerScrewerFrontAxisRef.NcToPlc.ActPos;
				lrStartPositionScrewerRear					:=	RollerScrewerRearAxisRef.NcToPlc.ActPos;
			END_IF	
			
	  			
//====================================				
		
	(*Zakręcanie*)
	E_RollerScrewer.eScrewing:
	
			mcScrewerFrontMoveVelocity.Velocity				:=	lrScrewerSpeed;
			mcScrewerRearMoveVelocity.Velocity				:=	lrScrewerSpeed;
			IF ABS(ABS(lrStartPositionScrewerFront)-ABS(RollerScrewerFrontAxisRef.NcToPlc.ActPos))>30 OR 
				ABS(ABS(lrStartPositionScrewerRear)-ABS(RollerScrewerRearAxisRef.NcToPlc.ActPos))>30
			THEN
				uiScrewingFrontTorqueControl					:=	INT_TO_UINT(iScrewerSetTorque+5)*10;
				uiScrewingRearTorqueControl						:=	INT_TO_UINT(iScrewerSetTorque+5)*10;
			ELSE
				uiScrewingFrontTorqueControl					:=	(INT_TO_UINT(iScrewerSetTorque+5)*10)+500;	
				uiScrewingRearTorqueControl						:=	(INT_TO_UINT(iScrewerSetTorque+5)*10)+500;
			END_IF
			mcScrewerFrontMoveVelocity.Direction				:=	MC_Direction.MC_Positive_Direction;
			mcScrewerRearMoveVelocity.Direction					:=	MC_Direction.MC_Positive_Direction;			
			IF tonTopActuatorDelayOff.Q THEN
				bPressingTopActuator					:=	FALSE; // Odcisniecie wczesniej niz zakręcanie
			END_IF
		
			IF tonTightScrewingTimer.Q THEN
				bPressingTopActuator					:=	FALSE;
				bPressingRollsActuator					:=	FALSE;
				mcScrewerFrontMoveVelocity.Execute			:=	FALSE;
				mcScrewerFrontSoftReset						(Axis:=RollerScrewerFrontAxisRef, Execute:= TRUE);
				mcScrewerRearMoveVelocity.Execute			:=	FALSE;
				mcScrewerRearSoftReset						(Axis:=RollerScrewerRearAxisRef, Execute:= TRUE);
				uiScrewingFrontTorqueControl					:=	0;
				uiScrewingRearTorqueControl					:=	0;			
				bScrewed								:=	TRUE;		
			END_IF
			IF tonPressingRollsReliseDelay.Q AND bScrewed THEN //200ms
				eRunningState							:=	E_RollerScrewer.eGoingUp;
			END_IF	
	

//====================================
						
	E_RollerScrewer.eGoingUp:
	
			mcScrewerFrontSoftReset							(Axis:=RollerScrewerFrontAxisRef, Execute:=TRUE);
			mcScrewerFrontStop.Execute						:=	FALSE;
			mcScrewerRearSoftReset							(Axis:=RollerScrewerRearAxisRef, Execute:=TRUE);
			mcScrewerRearStop.Execute						:=	FALSE;			
			IF bRollsUnPressedSensor AND bUnPressedTopSensor THEN
				eRunningState							:=	E_RollerScrewer.eDone;
			END_IF

	
//====================================	
		 
	E_RollerScrewer.eDone:
	
			bScrewed									:=	FALSE;
			bScrewFound									:=	FALSE;
			
			mcScrewerFrontSoftReset							(Axis:=RollerScrewerFrontAxisRef, Execute:=TRUE);
			mcScrewerFrontStop.Execute						:=	FALSE;
			mcScrewerRearSoftReset							(Axis:=RollerScrewerRearAxisRef, Execute:=TRUE);
			mcScrewerRearStop.Execute						:=	FALSE;
			uiScrewingFrontTorqueControl						:=	0;	
			uiScrewingRearTorqueControl						:=	0;				
			bCycleDone 									:= TRUE;
			eRunningState								:= E_RollerScrewer.eReady;
	

//====================================	
			
	E_RollerScrewer.eNotDone:
	
		bCycleNotDone 									:=	TRUE;
		eRunningState									:=	E_RollerScrewer.eReady;	
		mcScrewerFrontSoftReset								(Axis:=RollerScrewerFrontAxisRef, Execute:=TRUE);
		mcScrewerRearSoftReset								(Axis:=RollerScrewerRearAxisRef, Execute:=TRUE);	
	
END_CASE
END_ACTION

ACTION ServoFrontControlBlocks:
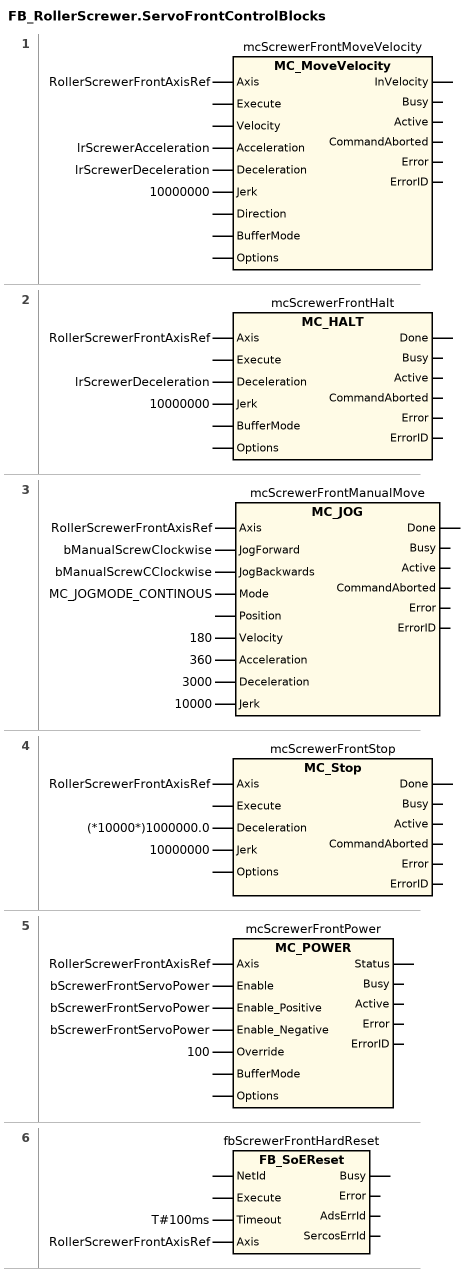
// NETWORK 1
mcScrewerFrontMoveVelocity(
    Axis := RollerScrewerFrontAxisRef,
    Acceleration := lrScrewerAcceleration,
    Deceleration := lrScrewerDeceleration,
    Jerk := 10000000); // MC_MoveVelocity

// NETWORK 2
mcScrewerFrontHalt(
    Axis := RollerScrewerFrontAxisRef,
    Deceleration := lrScrewerDeceleration,
    Jerk := 10000000); // MC_HALT

// NETWORK 3
mcScrewerFrontManualMove(
    Axis := RollerScrewerFrontAxisRef,
    JogForward := bManualScrewClockwise,
    JogBackwards := bManualScrewCClockwise,
    Mode := MC_JOGMODE_CONTINOUS,
    Velocity := 180,
    Acceleration := 360,
    Deceleration := 3000,
    Jerk := 10000); // MC_JOG

// NETWORK 4
mcScrewerFrontStop(Axis := RollerScrewerFrontAxisRef, Deceleration := (*10000*)1000000.0, Jerk := 10000000); // MC_Stop

// NETWORK 5
mcScrewerFrontPower(
    Axis := RollerScrewerFrontAxisRef,
    Enable := bScrewerFrontServoPower,
    Enable_Positive := bScrewerFrontServoPower,
    Enable_Negative := bScrewerFrontServoPower,
    Override := 100); // MC_POWER

// NETWORK 6
fbScrewerFrontHardReset(Timeout := T#100ms, Axis := RollerScrewerFrontAxisRef); // FB_SoEReset

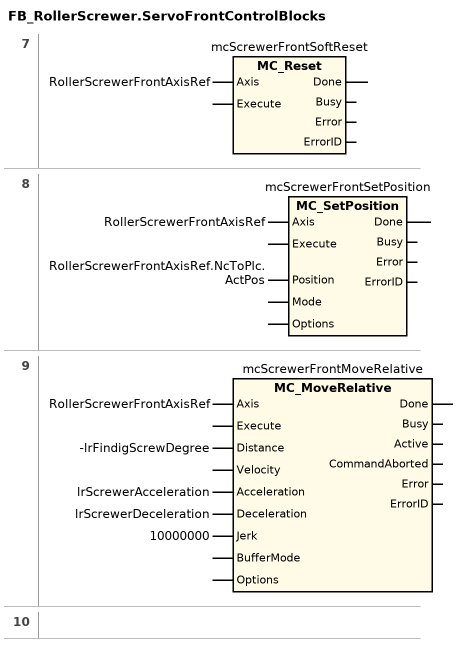
// NETWORK 7
mcScrewerFrontSoftReset(Axis := RollerScrewerFrontAxisRef); // MC_Reset

// NETWORK 8
mcScrewerFrontSetPosition(Axis := RollerScrewerFrontAxisRef, Position := RollerScrewerFrontAxisRef.NcToPlc.ActPos); // MC_SetPosition

// NETWORK 9
mcScrewerFrontMoveRelative(
    Axis := RollerScrewerFrontAxisRef,
    Distance := -lrFindigScrewDegree,
    Acceleration := lrScrewerAcceleration,
    Deceleration := lrScrewerDeceleration,
    Jerk := 10000000); // MC_MoveRelative

// NETWORK 10
END_ACTION

ACTION ServoRearControlBlocks:
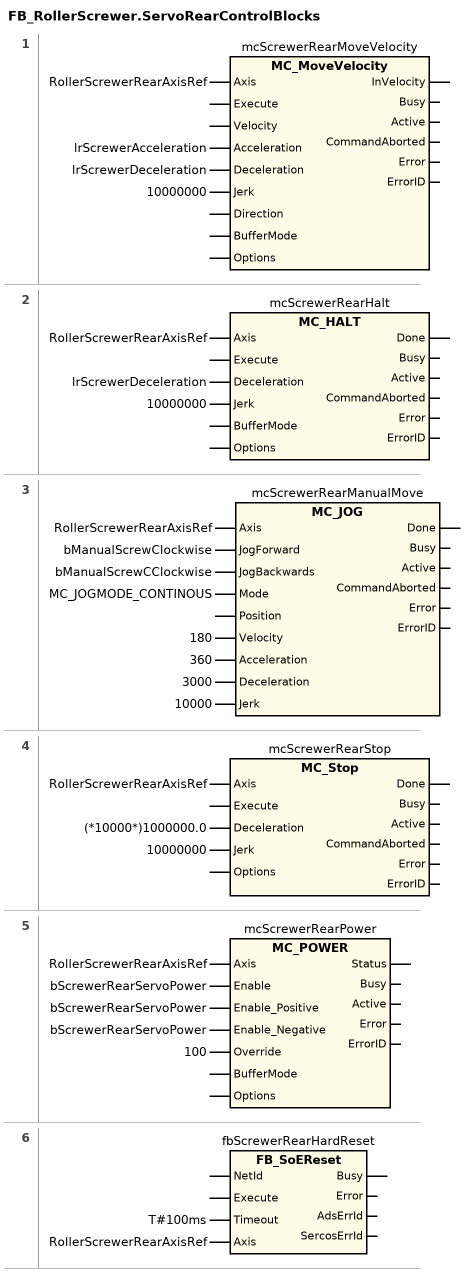
// NETWORK 1
mcScrewerRearMoveVelocity(
    Axis := RollerScrewerRearAxisRef,
    Acceleration := lrScrewerAcceleration,
    Deceleration := lrScrewerDeceleration,
    Jerk := 10000000); // MC_MoveVelocity

// NETWORK 2
mcScrewerRearHalt(Axis := RollerScrewerRearAxisRef, Deceleration := lrScrewerDeceleration, Jerk := 10000000); // MC_HALT

// NETWORK 3
mcScrewerRearManualMove(
    Axis := RollerScrewerRearAxisRef,
    JogForward := bManualScrewClockwise,
    JogBackwards := bManualScrewCClockwise,
    Mode := MC_JOGMODE_CONTINOUS,
    Velocity := 180,
    Acceleration := 360,
    Deceleration := 3000,
    Jerk := 10000); // MC_JOG

// NETWORK 4
mcScrewerRearStop(Axis := RollerScrewerRearAxisRef, Deceleration := (*10000*)1000000.0, Jerk := 10000000); // MC_Stop

// NETWORK 5
mcScrewerRearPower(
    Axis := RollerScrewerRearAxisRef,
    Enable := bScrewerRearServoPower,
    Enable_Positive := bScrewerRearServoPower,
    Enable_Negative := bScrewerRearServoPower,
    Override := 100); // MC_POWER

// NETWORK 6
fbScrewerRearHardReset(Timeout := T#100ms, Axis := RollerScrewerRearAxisRef); // FB_SoEReset

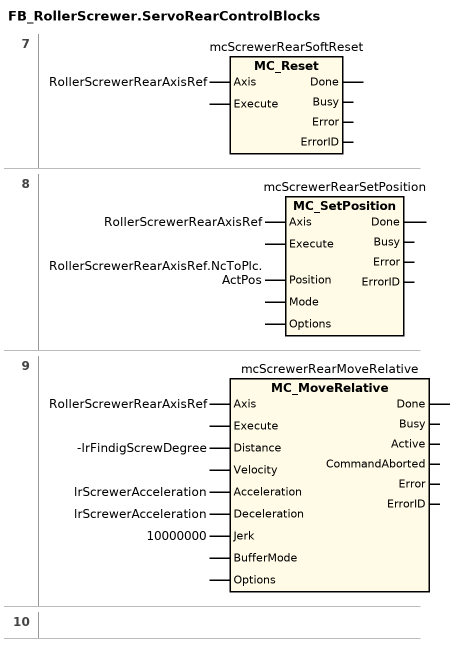
// NETWORK 7
mcScrewerRearSoftReset(Axis := RollerScrewerRearAxisRef); // MC_Reset

// NETWORK 8
mcScrewerRearSetPosition(Axis := RollerScrewerRearAxisRef, Position := RollerScrewerRearAxisRef.NcToPlc.ActPos); // MC_SetPosition

// NETWORK 9
mcScrewerRearMoveRelative(
    Axis := RollerScrewerRearAxisRef,
    Distance := -lrFindigScrewDegree,
    Acceleration := lrScrewerAcceleration,
    Deceleration := lrScrewerAcceleration,
    Jerk := 10000000); // MC_MoveRelative

// NETWORK 10
END_ACTION

ACTION Statistics:

rtrigCycleTimerRead(CLK:=(eRunningState=E_RollerScrewer.eDone) OR (eRunningState=E_RollerScrewer.eNotDone));
IF rtrigCycleTimerRead.Q THEN
	tCycleTime:=tonCycleTimer.ET;
END_IF
tonCycleTimer(IN:=eState>E_Station.eReady,PT:=T#1D);
END_ACTION

END_FUNCTION_BLOCK

(* stored: Version 1.2.0.0, ProductVersion 3.1.4026.13, FileIdentifier 61f333728d067ace1c11d39c72d0ab2f15fea670, FileSignature 585bece3c9ebdced7066f2962b33a7aee8206fe7b0876cd77711f71811f1b619d07412dfd0b94f4f3c916fb6eb9e57fab1dedcce39752c1eb5adc561d1ea1ff9fda3793fb1bdca23cf57d05157926eec0359e7d989d3219c5ca8893fd00cd7b0504b1149ee338c3e1368f1cc2581e311c834cf963e84d9e89db6baa13673707223fa79de6e90a41d71b83ee4f536c6367b389af7cee9c2c148a7fa86ee149c768db556ef953550b0616939dfc2a22fc81311cd3e0a6eb84f38ab547bfaeaf676acad49e9fa3488597b82c55a7f53f955ca99a8ec60e9ff5bcd95dcd4677824057ace67b615718170959b269a1e06e64f2f5101479e5a79645be27595dd6f6e2d
   POU FB_RollerScrewer: Id {626bd90c-8bf3-4131-98ce-3a74b2b41c80}, SpecialFunc None
   Action Control: Id {83df8312-ff43-460a-996d-8df3e9102e40}
   Action ErrorHandling: Id {b9fbb56c-2795-4b31-b607-694f0166ccce}
   Action HeightMotor: Id {ba3343f7-fff3-4f4a-89d1-f3eced85b074}
   Action Homing: Id {5455efc8-5ef5-4af1-8c49-7f5cd0b96e04}
   Action ManualMovements: Id {500cbaa6-9498-4e8e-8a5a-016682a915d6}
   Action Running: Id {a3a38408-5b15-456c-9eaa-233fc9e582ad}
   Action ServoFrontControlBlocks: Id {0a1d62b8-68ed-4a83-9cb5-935b6246f30e}
   Action ServoRearControlBlocks: Id {097374bd-bac7-4696-83e9-c0c15c0417c2}
   Action Statistics: Id {7ed1fa03-023a-4a5c-babe-eff2bfca8f6c} *)
